Universal Robots URScript: T013_qwen2.5-coder_32b_baseline_rep1.urscript

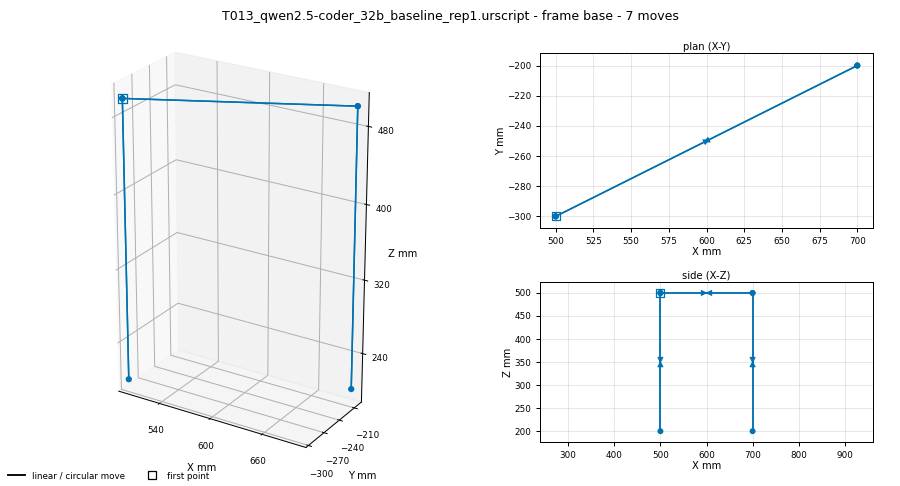
[picture p0: tool path of T013_qwen2.5-coder_32b_baseline_rep1.urscript in frame base, 7 of 9 moves have a stored position in this frame; points joined in program order, loops and branches not executed]
def task_t013():
    # Home position
    movej(get_inverse_kin([0, -90, 90, -90, 0, 0]), a=1.4, v=1.2)

    # Above staging area
    movel(p[0.5, -0.3, 0.5, 3.14, 0, 0], a=1.2, v=1.05)

    # Descend to pick position
    movel(p[0.5, -0.3, 0.2, 3.14, 0, 0], a=1.2, v=0.6)

    # Lift with suction cup engaged
    movel(p[0.5, -0.3, 0.5, 3.14, 0, 0], a=1.2, v=1.08)

    # Transit to pallet position
    movel(p[0.7, -0.2, 0.5, 3.14, 0, 0], a=1.2, v=1.15)

    # Descend to place position on pallet
    movel(p[0.7, -0.2, 0.2, 3.14, 0, 0], a=1.2, v=0.6)

    # Release suction cup and lift
    movel(p[0.7, -0.2, 0.5, 3.14, 0, 0], a=1.2, v=1.08)

    # Return to above staging area
    movel(p[0.5, -0.3, 0.5, 3.14, 0, 0], a=1.2, v=1.05)

    # Home position
    movej(get_inverse_kin([0, -90, 90, -90, 0, 0]), a=1.4, v=1.2)
end

task_t013()
